{attribute 'qualified_only'}
VAR_GLOBAL CONSTANT
	
	TOTAL_NUM_TESTS : INT := 70;
	
	SECTION1_NUM_DIG_TESTS : INT := 21;
	
	SECTION1_NUM_HMI_TESTS : INT := 2;
	
	SECTION2_NUM_DIG_TESTS : INT := 1;
	
	NUM_CONNECTIONS : INT := 30;
	
END_VAR

(* stored: Version 1.1.0.1, ProductVersion 3.1.4024.10
   GVL CONSTANTS: Id {46936124-0b4c-4191-8ea5-f9773d0032d0}, ParameterList True *)
